TYPE TcoInsightResults_v_5_x_x :
STRUCT	
	InspectionId: UINT;
	ResultCode: UINT;
	InspectionResults : ARRAY[0..TcoVisionParams.MAX_BYTE_ARRAY] OF BYTE;
END_STRUCT
END_TYPE

(* stored: Version 1.1.0.1, ProductVersion 3.1.4024.11
   DUT TcoInsightResults_v_5_x_x: Id {8dc06bb9-6b02-0926-1c36-0798891380d1} *)
